(* IEC 61131-3 sources: com.logicals.lc3.webinar/logicals_Lib_Webinar/logicals_Webinar_Basic_Lib/logicals_Lib/src_FB_FBD/Count, 4 files *)

(* ---- FB_lc_DecUDINT_FBD.iecfbd ---- *)
NAMESPACE com.logicals.Basic.Count
FUNCTION_BLOCK FB_lc_DecUDINT_FBD
  VAR_OUTPUT
    Cnt : UDINT := 0;
  END_VAR

  (*

    // Network 1:
    SUB(IN1 := Cnt, IN2 := 1, SUB => Cnt);

  *)

  @VF(104) : @E(Cnt), @R(600.0, 460.0, 90.0, 19.0);
  @VF(101) : @E(1), @R(600.0, 480.0, 40.0, 19.0), UDINT;
  @VF(102) : @E(Cnt), @R(1620.0, 460.0, 90.0, 19.0);
  @CF(100) : @R(330.0, 330.0, 430.0, 48.0), @T("Decrement UDINT-Variable to count events$N(starting with 0, count modulo EndVal=2^32)"), @POU;
  @CF(1) : @R(870.0, 330.0, 430.0, 48.0), @T("UDINT-Variable erniedrigen um Ereignisse zu zaehlen$N(Start mit 0, zaehlt modulo EndWert=2^32)"), @POU;
  @C(2) : @F(SUB), @R(720.0, 460.0, 40.0, 38.0), UDINT, @I(@N(IN1), @L(9.5)), @I(@N(IN2), @L(29.5)), @O(@N(SUB), @R(9.5));

  @G(3) :
     @L(@C(2).SUB, @VF(102).i)
    ;
  @G(4) :
     @L(@VF(104).o, @C(2).IN1)
    ;
  @G(5) :
     @L(@VF(101).o, @C(2).IN2)
    ;
END_FUNCTION_BLOCK
END_NAMESPACE

(* ---- FB_lc_DecUINT_FBD.iecfbd ---- *)
NAMESPACE com.logicals.Basic.Count
FUNCTION_BLOCK FB_lc_DecUINT_FBD
  VAR_OUTPUT
    Cnt : UINT := 0;
  END_VAR

  (*

    // Network 1:
    SUB(IN1 := Cnt, IN2 := 1, SUB => Cnt);

  *)

  @VF(104) : @E(Cnt), @R(600.0, 460.0, 90.0, 19.0);
  @VF(101) : @E(1), @R(600.0, 480.0, 40.0, 19.0), UINT;
  @VF(102) : @E(Cnt), @R(1620.0, 460.0, 90.0, 19.0);
  @CF(100) : @R(330.0, 330.0, 430.0, 48.0), @T("Decrement UINT-Variable to count events$N(starting with 0, count modulo 64K=2^16)"), @POU;
  @CF(1) : @R(870.0, 330.0, 430.0, 48.0), @T("UINT-Variable erniedrigen um Ereignisse zu zaehlen$N(Start mit 0, zaehlt modulo 64K=2^16)"), @POU;
  @C(2) : @F(SUB), @R(730.0, 460.0, 40.0, 38.0), UINT, @I(@N(IN1), @L(9.5)), @I(@N(IN2), @L(29.5)), @O(@N(SUB), @R(9.5));

  @G(3) :
     @L(@C(2).SUB, @VF(102).i)
    ;
  @G(4) :
     @L(@VF(104).o, @C(2).IN1)
    ;
  @G(5) :
     @L(@VF(101).o, @C(2).IN2)
    ;
END_FUNCTION_BLOCK
END_NAMESPACE

(* ---- FB_lc_IncUDINT_FBD.iecfbd ---- *)
NAMESPACE com.logicals.Basic.Count
FUNCTION_BLOCK FB_lc_IncUDINT_FBD
  VAR_OUTPUT
    Cnt : UDINT := 0;
  END_VAR

  (*

    // Network 1:
    ADD(IN1 := Cnt, IN2 := 1, ADD => Cnt);

  *)

  @C(103) : @F(ADD), @R(730.0, 460.0, 40.0, 38.0), UDINT, @I(@N(IN1), @L(9.5)), @I(@N(IN2), @L(29.5)), @O(@N(ADD), @R(9.5));
  @VF(104) : @E(Cnt), @R(600.0, 460.0, 90.0, 19.0);
  @VF(101) : @E(1), @R(600.0, 480.0, 40.0, 19.0), UDINT;
  @VF(102) : @E(Cnt), @R(1620.0, 460.0, 90.0, 19.0);
  @CF(100) : @R(330.0, 330.0, 430.0, 48.0), @T("Increment UDINT-Variable to count events$N(starting with 0, count modulo EndVal=2^32)"), @POU;
  @CF(1) : @R(870.0, 330.0, 430.0, 48.0), @T("UDINT-Variable erhoehen um Ereignisse zu zaehlen$N(Start mit 0, zaehlt modulo EndWert=2^32)"), @POU;

  @G(107) :
     @L(@VF(104).o, @C(103).IN1)
    ;
  @G(108) :
     @L(@VF(101).o, @C(103).IN2)
    ;
  @G(106) :
     @L(@C(103).ADD, @VF(102).i)
    ;
END_FUNCTION_BLOCK
END_NAMESPACE

(* ---- FB_lc_IncUINT_FBD.iecfbd ---- *)
NAMESPACE com.logicals.Basic.Count
FUNCTION_BLOCK FB_lc_IncUINT_FBD
  VAR_OUTPUT
    Cnt : UINT := 0;
  END_VAR

  (*

    // Network 1:
    ADD(IN1 := Cnt, IN2 := 1, ADD => Cnt);

  *)

  @C(103) : @F(ADD), @R(730.0, 460.0, 40.0, 38.0), UINT, @I(@N(IN1), @L(9.5)), @I(@N(IN2), @L(29.5)), @O(@N(ADD), @R(9.5));
  @VF(104) : @E(Cnt), @R(600.0, 460.0, 90.0, 19.0);
  @VF(101) : @E(1), @R(600.0, 480.0, 40.0, 19.0), UINT;
  @VF(102) : @E(Cnt), @R(1620.0, 460.0, 90.0, 19.0);
  @CF(100) : @R(330.0, 330.0, 430.0, 48.0), @T("Increment UINT-Variable to count events$R$N(starting with 0, count modulo 64K=2^16)"), @POU;
  @CF(1) : @R(870.0, 330.0, 430.0, 48.0), @T("UINT-Variable erhoehen um Ereignisse zu zaehlen$N(Start mit 0, zaehlt modulo 64K=2^16)"), @POU;

  @G(107) :
     @L(@VF(104).o, @C(103).IN1)
    ;
  @G(108) :
     @L(@VF(101).o, @C(103).IN2)
    ;
  @G(106) :
     @L(@C(103).ADD, @VF(102).i)
    ;
END_FUNCTION_BLOCK
END_NAMESPACE
